TYPE ST_PistonRange :
STRUCT
	fPistonPosMax : REAL := 0.5;
	fPistonPosMin : REAL := 0.0;
END_STRUCT
END_TYPE

(* stored: Version 1.1.0.1, ProductVersion 3.1.4024.10
   DUT ST_PistonRange: Id {2ff82653-f802-433f-9d13-ab0873d2b7c8} *)
